FUNCTION mmHgToPascal : Pascal
VAR_INPUT
     pressure : mmHg;
END_VAR

mmHgToPascal._ := pressure._ * 133322;

END_FUNCTION

(* stored: Version 1.1.0.1, ProductVersion 3.1.4024.4
   POU mmHgToPascal: Id {a6985b3d-4ca0-4ab1-9135-42f98adb9f8f}, SpecialFunc None *)
